Universal Robots PolyScope program: p12kine.urp

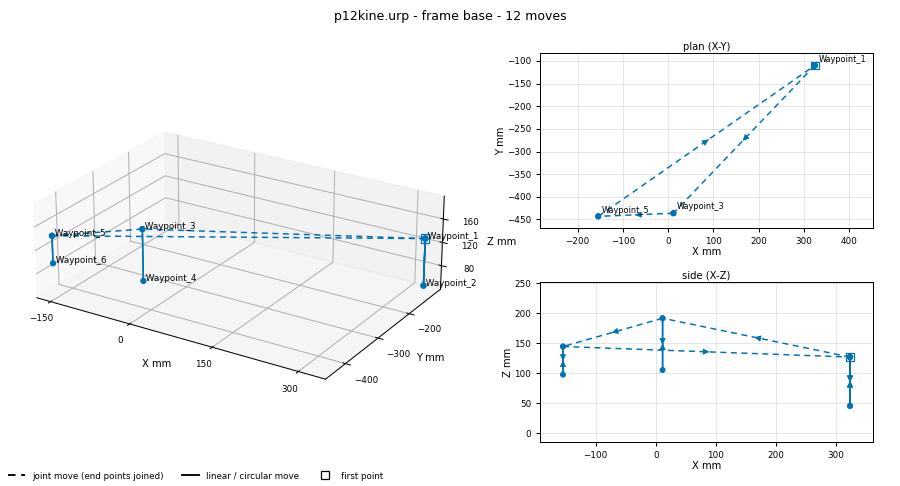
[picture p0: tool path of p12kine.urp in frame base, 12 of 12 moves have a stored position in this frame; points joined in program order, loops and branches not executed]
Program p12kine (installation=default directory=/programs createdIn=5.14.5 lastSavedIn=5.14.5 robotSerialNumber=20195300809)
Calibrated DH parameters: a=[-0.000085, -0.20076, -0.212369, 0.000121, -0.000118, 0]; d=[0.15185, -26.306375, 24.753047, 1.684739, 0.085386, 0.092088]; alpha=[1.572149, -0.00522, -0.011864, 1.571339, -1.571085, 0]; deltaTheta=[0, 0.599885, -0.513355, -0.086555, 0.000006, 0]
InitVariablesNode
Robot Program (runOnlyOnce=false)
  URCap Gripper (Robotiq_Grippers, Robotiq Inc.) dataModel(position=0.0, force=0.0, speed=100.0, positionInDouble=0.0, forceInDouble=0.0, speedInDouble=100.0, slaveIds=[9], blocking=true)
  Wait Sleep waitTime=1
  MoveJ speed 60 deg/s, acceleration 80 deg/s^2 (useActiveTCP=true) feature=Base
    Waypoint Waypoint_1: TCP in base x=323.542 y=-110.249 z=127.21 mm, rx=2.9911 ry=0.2085 rz=0.059 rad; joints [10.735, -88.214, -93.185, -87.344, 81.034, -87.032] deg; TCP offset x=0 y=0 z=174 mm, rx=0 ry=0 rz=0 rad
  MoveL speed 250 mm/s, acceleration 1200 mm/s^2 (useActiveTCP=true) feature=Base
    Waypoint Waypoint_2: TCP in base x=323.536 y=-110.243 z=45.884 mm, rx=2.9911 ry=0.2086 rz=0.059 rad; joints [10.838, -92.596, -111.336, -64.789, 81.055, -87.182] deg
    URCap Gripper (Robotiq_Grippers, Robotiq Inc.) dataModel(position=100.0, force=0.0, speed=100.0, positionInDouble=100.0, forceInDouble=0.0, speedInDouble=100.0, slaveIds=[9], blocking=true)
    Wait Sleep waitTime=1
    Waypoint Waypoint_1: TCP in base x=323.542 y=-110.249 z=127.21 mm, rx=2.9911 ry=0.2085 rz=0.059 rad; joints [10.735, -88.214, -93.185, -87.344, 81.034, -87.032] deg
  MoveJ speed 60 deg/s, acceleration 80 deg/s^2 (useActiveTCP=true) feature=Base
    Waypoint Waypoint_3: TCP in base x=11.501 y=-436.256 z=191.852 mm, rx=3.0173 ry=-0.0326 rz=0.115 rad; joints [-72.496, -112.998, -48.153, -100.816, 91.249, -160.615] deg
  MoveL speed 250 mm/s, acceleration 1200 mm/s^2 (useActiveTCP=true) feature=Base
    Waypoint Waypoint_4: TCP in base x=11.5 y=-436.24 z=105.662 mm, rx=3.0175 ry=-0.0326 rz=0.1148 rad; joints [-72.437, -110.505, -75.177, -76.304, 91.231, -160.847] deg
    URCap Gripper (Robotiq_Grippers, Robotiq Inc.) dataModel(position=0.0, force=0.0, speed=100.0, positionInDouble=0.0, forceInDouble=0.0, speedInDouble=100.0, slaveIds=[9], blocking=true)
    Wait Sleep waitTime=1
    Waypoint Waypoint_3: TCP in base x=11.501 y=-436.256 z=191.852 mm, rx=3.0173 ry=-0.0326 rz=0.115 rad; joints [-72.496, -112.998, -48.153, -100.816, 91.249, -160.615] deg
    Set DigitalOutput pin=digital_out[0]; digitalValue=1
  Wait DigitalInput pin=digital_in[0]; digitalValue=0
  Set IncrementVariable installationVariable=cont
  MoveJ speed 60 deg/s, acceleration 80 deg/s^2 (useActiveTCP=true) feature=Base
    Waypoint Waypoint_5: TCP in base x=-154.347 y=-443.128 z=144.76 mm, rx=3.0891 ry=0.1107 rz=-0.0972 rad; joints [-91.171, -125.231, -39.384, -102.391, 85.815, -184.837] deg
  MoveL speed 250 mm/s, acceleration 1200 mm/s^2 (useActiveTCP=true) feature=Base
    Waypoint Waypoint_6: TCP in base x=-154.368 y=-443.108 z=97.918 mm, rx=3.0891 ry=0.1107 rz=-0.0973 rad; joints [-91.155, -123.164, -55.535, -88.299, 85.793, -184.984] deg
    URCap Gripper (Robotiq_Grippers, Robotiq Inc.) dataModel(position=100.0, force=0.0, speed=100.0, positionInDouble=100.0, forceInDouble=0.0, speedInDouble=100.0, slaveIds=[9], blocking=true)
    Waypoint Waypoint_5: TCP in base x=-154.347 y=-443.128 z=144.76 mm, rx=3.0891 ry=0.1107 rz=-0.0972 rad; joints [-91.171, -125.231, -39.384, -102.391, 85.815, -184.837] deg
  If cont≤2
    MoveJ speed 60 deg/s, acceleration 80 deg/s^2 (useActiveTCP=true) feature=Base
      Waypoint Waypoint_1: TCP in base x=323.542 y=-110.249 z=127.21 mm, rx=2.9911 ry=0.2085 rz=0.059 rad; joints [10.735, -88.214, -93.185, -87.344, 81.034, -87.032] deg
    MoveL speed 250 mm/s, acceleration 1200 mm/s^2 (useActiveTCP=true) feature=Base
      Waypoint Waypoint_2: TCP in base x=323.536 y=-110.243 z=45.884 mm, rx=2.9911 ry=0.2086 rz=0.059 rad; joints [10.838, -92.596, -111.336, -64.789, 81.055, -87.182] deg
      URCap Gripper (Robotiq_Grippers, Robotiq Inc.) dataModel(position=0.0, force=0.0, speed=100.0, positionInDouble=0.0, forceInDouble=0.0, speedInDouble=100.0, slaveIds=[9], blocking=true)
      Wait Sleep waitTime=1
      Waypoint Waypoint_1: TCP in base x=323.542 y=-110.249 z=127.21 mm, rx=2.9911 ry=0.2085 rz=0.059 rad; joints [10.735, -88.214, -93.185, -87.344, 81.034, -87.032] deg
  Else 
    Script: 
    Set Undefined
